FUNCTION_BLOCK MSLAVE_8_tcp (* 8-Channel Modbus TCP Slave Interface Block *)
  (* Version 1.0, AN, SWDC RTSoft *)
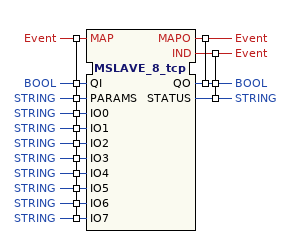
  EVENT_INPUT
    MAP WITH QI, PARAMS, IO0, IO1, IO2, IO3, IO4, IO5, IO6, IO7; (* Initialization Request *)
  END_EVENT
  EVENT_OUTPUT
    MAPO WITH QO; (* Initialization Confirm *)
    IND WITH QO, STATUS; (* Execution Confirm *)
  END_EVENT
  VAR_INPUT
    QI : BOOL; (* Event Input Qualifier *)
    PARAMS : STRING; (* Initialization Parameters *)
    IO0 : STRING; (* Input Output 0 *)
    IO1 : STRING; (* Input Output 1 *)
    IO2 : STRING; (* Input Output 2 *)
    IO3 : STRING; (* Input Output 3 *)
    IO4 : STRING; (* Input Output 4 *)
    IO5 : STRING; (* Input Output 5 *)
    IO6 : STRING; (* Input Output 6 *)
    IO7 : STRING; (* Input Output 7 *)
  END_VAR
  VAR_OUTPUT
    QO : BOOL; (* Event Output Qualifier *)
    STATUS : STRING; (* Service Status *)
  END_VAR
END_FUNCTION_BLOCK
